PROGRAM C_1_PRG_MainHMI
VAR
	
	bResetTest				: BOOL;
	i						: DINT;
	n						: DINT;//TABLE INDEX
	bProcessDoorClosed		: BOOL;
	srRejectChuteFull		: SR; 

END_VAR

a_ACT_MachineStatusBaner();
b_ACT_Timers();
c_ACT_IO();

bEnableSettings				:= (stMachineStatus.eMachineState = E_MachineState.STOPPED);
bOpenRejectDialog			:= bRejectPartDialog[0] OR bRejectPartDialog[1] OR bRejectPartDialog[2];

bProcessDoorClosed			:= dw_T05_EL1918.iProcessDoorClosed1 AND dw_T05_EL1918.iProcessDoorClosed2 AND dw_T05_EL1918.iProcessDoorFB;

srRejectChuteFull(SET1 := stStationEvents[0].aEvents[18].bEventTimer.Q, RESET := bEmptyRejectChuteAcknowledge AND NOT dw_T08_EL1809.iRejectSensor , Q1 => bEmptyRejectChute);

bEnable_VacuumCylinder[1]				:= bProcessDoorClosed;
bEnable_VacuumCylinder[2]				:= bProcessDoorClosed;

IF NOT stMachineStatus.bManualMode THEN
	
	bHoldPart1							:= FALSE;
	bHoldPart2							:= FALSE;

END_IF

ACTION a_ACT_MachineStatusBaner:
//Machine status banner action
//SYSTEM POWER UP
IF stMachineStatus.bSystemPowerUp THEN	
	stStatusBanner.sMachineStatusText 							:= 'SYSTEM POWER UP';	
	stStatusBanner.nMachineStatusColour 						:= nWHITE;
	stStatusBanner.nMachineStatusTxtCol 						:= nBLACK;
	stStatusBanner.sBannerBckColor 								:= sWHITE;
	stStatusBanner.sBannerTextColor 							:= sBLACK;
END_IF

(* SYSTEM INITIALISING *)
IF stMachineStatus.bInitialising THEN	
	stStatusBanner.sMachineStatusText 							:= 'SYSTEM INITIALIZING';		
	stStatusBanner.nMachineStatusColour 						:= nYELLOW;
	stStatusBanner.nMachineStatusTxtCol 						:= nBLACK;
	stStatusBanner.sBannerBckColor 								:= sYELLOW;
	stStatusBanner.sBannerTextColor 							:= sBLACK;
END_IF

(* SAFETY *)
IF stMachineStatus.bSafety THEN	
	stStatusBanner.sMachineStatusText 							:= 'SYSTEM INITIALIZING';		
	stStatusBanner.nMachineStatusColour 						:= nYELLOW;
	stStatusBanner.nMachineStatusTxtCol 						:= nBLACK;
	stStatusBanner.sBannerBckColor 								:= sYELLOW;
	stStatusBanner.sBannerTextColor 							:= sBLACK;
END_IF


(* SYSTEM READY TO START FLASH ON *)
IF stMachineStatus.bReadyToStart AND stPuls.bFlash1Hz THEN
	stStatusBanner.sMachineStatusText 							:= 'SYSTEM READY TO START';		
	stStatusBanner.nMachineStatusColour 						:= nGREEN;
	stStatusBanner.nMachineStatusTxtCol 						:= nWHITE;
	stStatusBanner.sBannerBckColor 								:= sGREEN;
	stStatusBanner.sBannerTextColor 							:= sWHITE;
ELSIF stMachineStatus.bReadyToStart AND NOT stPuls.bFlash1Hz THEN	
	stStatusBanner.sMachineStatusText 							:= 'SYSTEM READY TO START';		
	stStatusBanner.nMachineStatusColour 						:= nWHITE;
	stStatusBanner.nMachineStatusTxtCol 						:= nGREEN;
	stStatusBanner.sBannerBckColor 								:= sWHITE;
	stStatusBanner.sBannerTextColor 							:= sGREEN;
END_IF

(* SYSTEM AUTO CYCLE *)
IF stMachineStatus.bAutoCycle THEN	
	stStatusBanner.sMachineStatusText 							:= 'SYSTEM AUTO CYCLE';		
	stStatusBanner.nMachineStatusColour 						:= nGREEN;
	stStatusBanner.nMachineStatusTxtCol 						:= nWHITE;
	stStatusBanner.sBannerBckColor 								:= sGREEN;
	stStatusBanner.sBannerTextColor 							:= sWHITE;	
END_IF

(* STOPPING *)
IF stMachineStatus.bStopping AND stPuls.bFlash1Hz THEN	
	stStatusBanner.sMachineStatusText 							:= 'STOPPING';		
	stStatusBanner.nMachineStatusColour 						:= nBLACK;
	stStatusBanner.nMachineStatusTxtCol 						:= nWHITE;
	stStatusBanner.sBannerBckColor 								:= sBLACK;
	stStatusBanner.sBannerTextColor 							:= sWHITE;	
ELSIF stMachineStatus.bStopping AND NOT stPuls.bFlash1Hz THEN	
	stStatusBanner.sMachineStatusText 							:= 'STOPPING';		
	stStatusBanner.nMachineStatusColour 						:= nWHITE;
	stStatusBanner.nMachineStatusTxtCol 						:= nBLACK;
	stStatusBanner.sBannerBckColor 								:= sWHITE;
	stStatusBanner.sBannerTextColor 							:= sBLACK;	
END_IF

(*STOPPED *)
IF stMachineStatus.bStopped THEN	
	stStatusBanner.sMachineStatusText 							:= 'CYCLE STOPPED';		
	stStatusBanner.nMachineStatusColour 						:= nBLACK;
	stStatusBanner.nMachineStatusTxtCol 						:= nWHITE;
	stStatusBanner.sBannerBckColor 								:= sBLACK;
	stStatusBanner.sBannerTextColor 							:= sWHITE;	
END_IF

(* FAULT FLASH ON *)
IF stMachineStatus.bFault AND stPuls.bFlash1Hz THEN	
	stStatusBanner.sMachineStatusText 							:= 'FAULT';		
	stStatusBanner.nMachineStatusColour 						:= nRED;
	stStatusBanner.nMachineStatusTxtCol 						:= nWHITE;
	stStatusBanner.sBannerBckColor 								:= sRED;
	stStatusBanner.sBannerTextColor 							:= sWHITE;	
ELSIF stMachineStatus.bFault AND NOT stPuls.bFlash1Hz THEN	
	stStatusBanner.sMachineStatusText 							:= 'FAULT';		
	stStatusBanner.nMachineStatusColour 						:= nWHITE;
	stStatusBanner.nMachineStatusTxtCol 						:= nBLACK;
	stStatusBanner.sBannerBckColor 								:= sWHITE;
	stStatusBanner.sBannerTextColor 							:= sBLACK;	
END_IF

(* MANUAL MODE *)
IF stMachineStatus.bManualMode THEN	
	stStatusBanner.sMachineStatusText 							:= 'MANUAL MODE';		
	stStatusBanner.nMachineStatusColour 						:= nBLUE;
	stStatusBanner.nMachineStatusTxtCol 						:= nWHITE;
	stStatusBanner.sBannerBckColor 								:= sBLUE;
	stStatusBanner.sBannerTextColor 							:= sWHITE;	
END_IF
END_ACTION

ACTION b_ACT_Timers:

stTimers.tAutoCycleTimeOut		:= DINT_TO_TIME(stTimers.nAutoCycleTimeOut * 1000) ;
stTimers.tDoorOpenedSignal		:= DINT_TO_TIME(stTimers.nDoorOpenedSignal * 1000) ;
stTimers.tStation1TimeOut		:= DINT_TO_TIME(stTimers.nStation1TimeOut * 1000) ;
stTimers.tStation2TimeOut		:= DINT_TO_TIME(stTimers.nStation2TimeOut * 1000) ;
stTimers.tStation3TimeOut		:= DINT_TO_TIME(stTimers.nStation3TimeOut * 1000) ;
stTimers.tTwoHandsSignal		:= DINT_TO_TIME(stTimers.nTwoHandsSignal * 1000) ;
stTimers.tHeightTest			:= DINT_TO_TIME(stTimers.nHeightTest * 1000) ;
stTimers.tAutoCycleIDLETimeOut			:= DINT_TO_TIME(stTimers.nAutoCycleIDLETimeOut * 1000) ;
END_ACTION

ACTION c_ACT_IO:
dw_T09_EL2809.qPanelLightLED				:= bLightsOnOff;
END_ACTION

END_PROGRAM

(* stored: Version 1.1.0.1, ProductVersion 3.1.4026.18
   POU C_1_PRG_MainHMI: Id {74beadf6-2d48-457c-a28f-741842f8514e}, SpecialFunc None
   Action a_ACT_MachineStatusBaner: Id {0dc7bcd3-753a-4f06-be0f-fec0a8964021}
   Action b_ACT_Timers: Id {66f47bca-34fc-4901-8482-712d454221dd}
   Action c_ACT_IO: Id {5594a5d6-af1e-4a8b-85d6-f9bf1b336af1} *)
